// SIMATIC STEP 7 (V5.x) project utf
// CPU: CPU 315-2PN/DP
// station: Hardware
// station: SIMATIC 300
// station: P_ADR_BUS
// program: S7-Programm

SYMBOL_TABLE
"_tl_global"	DB 500	DB 500	// Global variables for tests
"_tl_const"	DB 501	DB 501	// Global constants
"TestCase"	FB 500	FB 500	// Test case and execution information
"_tl_assertStats"	UDT 500	UDT 500	// Assertion intermediary states data structure
END_SYMBOL_TABLE

TYPE "_tl_assertStats"	// UDT 500
AUTHOR : FlorianH
FAMILY : APTest
NAME : TL_stats
VERSION : 1.0
  STRUCT
   Trig : BOOL ;	// Assertion triggered
   Done : BOOL ;	// Assertion done
   Success : BOOL ;	// Assertion result
  END_STRUCT ;	
END_TYPE

FUNCTION_BLOCK "TestCase"	// FB 500
TITLE = APTest TestCase program
AUTHOR : FlorianH
FAMILY : APTest
NAME : TestCase
VERSION : 1.0
VAR
  testLog : ARRAY  [1 .. 63 ] OF STRING  [25 ];
  Tests : ARRAY  [0 .. 9 ] OF STRUCT
   TestName : STRING  [10 ];	//Name of the test
   ExecCounter : BYTE ;	//0 = no executions jet, > no OF exec
   StartTime : TIME ;	//TIME in ms OF the start OF the test, based on TIME()
   EndTime : DWORD ;	//sets a minimum TIME FOR the test step TO survive, also timeout
   State : BYTE ;	//Test CASE AND test state
   Result : BYTE ;	//Result, _tlState
   TestCounter : BYTE ;	//Test Number, in the test CASE
   TestStep : BYTE ;	//Actual test step
   TestCount : BYTE  := B#16#1;	//Total tests FOR this tc
   TestSteps : BYTE  := B#16#1;	//Total test steps
   AssertStats : ARRAY  [0 .. 3 ] OF //assert memory
   STRUCT 	//assert memory
    Trig : BOOL ;	// Assertion triggered
    Done : BOOL ;	// Assertion done
    Success : BOOL ;	// Assertion result
   END_STRUCT ;
  END_STRUCT ;
END_VAR
BEGIN
// body was compiled from an SCL source; compiled code not shown
END_FUNCTION_BLOCK

ORGANIZATION_BLOCK OB 1
TITLE = "Main Program Sweep (Cycle)"
VERSION : 0.1
VAR_TEMP
  OB1_EV_CLASS : BYTE ;	//Bits 0-3 = 1 (Coming event), Bits 4-7 = 1 (Event class 1)
  OB1_SCAN_1 : BYTE ;	//1 (Cold restart scan 1 of OB 1), 3 (Scan 2-n of OB 1)
  OB1_PRIORITY : BYTE ;	//Priority of OB Execution
  OB1_OB_NUMBR : BYTE ;	//1 (Organization block 1, OB1)
  OB1_RESERVED_1 : BYTE ;	//Reserved for system
  OB1_RESERVED_2 : BYTE ;	//Reserved for system
  OB1_PREV_CYCLE : INT ;	//Cycle time of previous OB1 scan (milliseconds)
  OB1_MIN_CYCLE : INT ;	//Minimum cycle time of OB1 (milliseconds)
  OB1_MAX_CYCLE : INT ;	//Maximum cycle time of OB1 (milliseconds)
  OB1_DATE_TIME : DATE_AND_TIME ;	//Date and time OB1 started
END_VAR
BEGIN
// (block stored without names or comments; labels and parameter names are numbered)
END_ORGANIZATION_BLOCK
